// TwinCAT 3 PLC project Main
// ProgramVersion: 3.1.4023.0
// libraries:
//   Tc2_Standard, * (Beckhoff Automation GmbH)
//   Tc2_System, * (Beckhoff Automation GmbH)
//   Tc3_JsonXml, * (Beckhoff Automation GmbH)
//   Tc3_Module, * (Beckhoff Automation GmbH)
// project tree:
//   / PlcTask.TcTTO
//   POUs/ FB_CountStructElements.TcPOU, MAIN.TcPOU, ST_Employee.TcDUT
// real-time tasks:
//   TASK PlcTask: cycle T#10ms, priority 20, ADS port 350

CONFIGURATION Main
    RESOURCE PLC ON TwinCAT3
        TASK PlcTask(INTERVAL := T#10ms, PRIORITY := 20);
        PROGRAM MAIN WITH PlcTask : MAIN;
    END_RESOURCE
END_CONFIGURATION

// ---- POUs/ST_Employee.TcDUT
TYPE ST_Employee :
STRUCT
	sName: STRING; 	  
	nEmployeeID : INT;
	nAge : INT;
END_STRUCT
END_TYPE

// ---- POUs/MAIN.TcPOU
PROGRAM MAIN
VAR
	stEmployee : ST_Employee;
	nStEmployeeElementCount : ULINT;
	fbCountStructElements : FB_CountStructElements;
END_VAR

fbCountStructElements(stAny := stEmployee, nElementsCount=> nStEmployeeElementCount );

END_PROGRAM

// ---- POUs/FB_CountStructElements.TcPOU
FUNCTION_BLOCK FB_CountStructElements
VAR_INPUT
	stAny : ANY;
END_VAR
VAR_OUTPUT
	nElementsCount : ULINT;
END_VAR
VAR
	transform : FB_JsonReadWriteDataType;
	datatypeName : STRING;
	jsonStringLength : UDINT;
	pJsonString : POINTER TO STRING;
	parser : FB_JsonDomParser;
	jsonDocument : SJsonValue;
	currentMember : SJsonValue;
	memberEnd : SJsonValue;
END_VAR

nElementsCount := 0;

datatypeName := transform.GetDataTypeNameByAddress(DINT_TO_UDINT(stAny.diSize),stAny.pValue);
jsonStringLength := transform.GetSizeJsonStringFromSymbol(datatypeName,DINT_TO_UDINT(stAny.diSize),stAny.pValue);

IF jsonStringLength = 0 THEN 
	RETURN;
END_IF

pJsonString := __NEW(BYTE,jsonStringLength);
transform.CopyJsonStringFromSymbol(datatypeName,DINT_TO_UDINT(stAny.diSize), stAny.pValue,pJsonString^,jsonStringLength);

jsonDocument := parser.ParseDocument(pJsonString^);
currentMember := parser.MemberBegin(jsonDocument);
memberEnd := parser.MemberEnd(jsonDocument);

WHILE currentMember <> memberEnd DO
	nElementsCount := nElementsCount + 1;
 	currentMember := parser.NextMember(currentMember);
END_WHILE

parser.NewDocument();
__DELETE(pJsonString);

END_FUNCTION_BLOCK
